PROGRAM MAIN
VAR
	
	MasterAxis		: MasterAxisControl;
	SlaveAxis		: SlaveAxisControl;
	Length			: LREAL := 200;
	Width			: LREAL := 40;
	Size			: LREAL := 80;
	xStart			: LREAL := 800;
	yStart			: LREAL := 400;
	State			: BYTE;
	
	Kinematic		: KinematicControl;
	
END_VAR

MasterAxis.CyclicUpdate();
SlaveAxis.CyclicUpdate();

MasterAxis.LengthOfShaft		 	:= Length;
MasterAxis.WidthOfShaft 			:= Width;
MasterAxis.AxisSize 				:= Size;
MasterAxis.XCoord 					:= xStart;
MasterAxis.YCoord 					:= yStart;

SlaveAxis.LengthOfShaft 			:= 150;
SlaveAxis.WidthOfShaft 				:= 60;
SlaveAxis.PreviousWidthOfShaft 		:= MasterAxis.WidthOfShaft;
SlaveAxis.PreviousAnglePosition 	:= MasterAxis.AnglePosition;
SlaveAxis.PreviousLengthOfShaft 	:= MasterAxis.LengthOfShaft;

SlaveAxis.PreviousXCoordGlobal 		:= MasterAxis.XCoord;
SlaveAxis.PreviousYCoordGlobal 		:= MasterAxis.YCoord;
SlaveAxis.PreviousXCoordRelative	:= MasterAxis.XCoord;
SlaveAxis.PreviousYCoordRelative	:= MasterAxis.YCoord;

CASE State OF
	
	0:
		IF MasterAxis.PowerOn() AND_THEN SlaveAxis.PowerOn() THEN
			State := 1;
		END_IF
		
	1:
		MasterAxis.MoveRelative(Position := 360, Velocity := 10);
	
END_CASE




Kinematic.CyclicUpdate();

END_PROGRAM

(* stored: Version 1.1.0.1, ProductVersion 3.1.4024.12
   POU MAIN: Id {1942bbfe-1c38-434d-8bb8-ce0fafb3b662}, SpecialFunc None *)
